INTERFACE IPLCopenCallStatus EXTENDS __SYSTEM.IQueryInterface

PROPERTY Abort : bool
GET
END_GET
SET
END_SET
END_PROPERTY

PROPERTY RemoteStatus : PLCopenStatusBase
GET
END_GET
SET
END_SET
END_PROPERTY

END_INTERFACE

(* stored: Version 1.1.0.1
   Itf IPLCopenCallStatus: Id {60f3b750-fcda-423b-b14b-4ab6a5b83007}
   Property Abort: Id {e3fd7230-b538-4c9e-9d21-fdf83ee0041b}
   Get Get: Id {c13334cc-4ce3-4ae4-ba07-5566ef4ed077}
   Set Set: Id {0f7f4071-2fa0-473a-b32d-6402c6d8e632}
   Property RemoteStatus: Id {6834da51-f1de-4461-86ce-4cf82752cb59}
   Get Get: Id {50c02346-7f00-4c9c-8cf9-194c91ed90ea}
   Set Set: Id {9f4e0d74-b30f-4fda-8eeb-5e79f6183d14} *)
